Universal Robots PolyScope program: sand1.urp

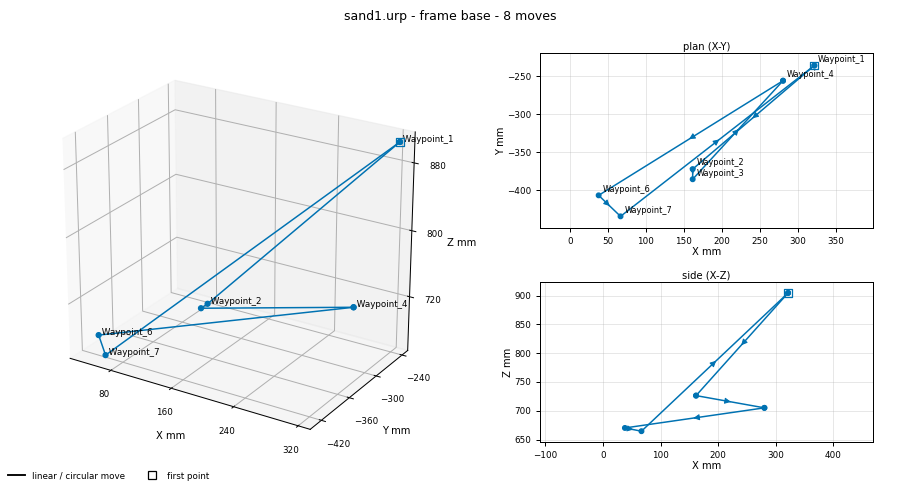
[picture p0: tool path of sand1.urp in frame base, 8 of 8 moves have a stored position in this frame; points joined in program order, loops and branches not executed]
Program sand1 (installation=default directory=/programs/archive createdIn=5.11.5.1010327 lastSavedIn=5.11.5.1010327 robotSerialNumber=20215500677)
Calibrated DH parameters: a=[0.000204, -0.239222, -0.391845, -0.000001, 0.000022, 0]; d=[0.162722, -355.808559, 353.37206, 2.570385, 0.099741, 0.099629]; alpha=[1.571124, 0.000988, 0.008295, 1.568963, -1.570303, 0]; deltaTheta=[0, -0.973091, 7.204745, 0.05153, 0, 0]
Robot Program (runOnlyOnce=true)
  MoveL speed 250 mm/s, acceleration 1200 mm/s^2 (useActiveTCP=true) feature=Base
    Waypoint Waypoint_1: TCP in base x=321.303 y=-235.884 z=904.602 mm, rx=1.6587 ry=-0.1473 rz=0.1861 rad; joints [-0.443, -84.298, -49.771, -109.018, 6.234, 255.071] deg
    Waypoint Waypoint_2: TCP in base x=161.455 y=-371.962 z=726.332 mm, rx=1.5708 ry=0 rz=0 rad; joints [-34.424, -75.969, -96.664, -7.98, 34.505, 180.726] deg
    Waypoint Waypoint_3: TCP in base x=161.455 y=-385.282 z=726.331 mm, rx=1.5708 ry=0 rz=0 rad; joints [-36.543, -77.681, -95.379, -7.51, 36.62, 180.691] deg
    SuppressedNode
      URCap Find Surface (Robotiq_Copilot, Robotiq Inc.) dataModel(NodeInitializedKey=true, WaitForSteadyWrenchOptionKey=false, ls_force=10.0, ls_distance=100.0, ls_speed=5.0, ls_if_distance=false, ls_if_force=false, ZeroSensorBeforeKey=true); state(isChildrenLocked=true)
        'Add Stop conditions from the Find Surface node'
    SuppressedNode
      Point_2 := Joint_6_nameget_actual_tcp_pose()
    URCap Finishing Tool Control (Robotiq_Copilot, Robotiq Inc.) dataModel(ToolOutputNameKey=digital_out[0], HackTriggeringContributionIsDefinedMethodKey=true)
    URCap Force Control (Robotiq_Copilot, Robotiq Inc.) dataModel(NodeInitializedKey=true, force_x=0, force_y=0, force_mx=0, force_my=0, force_mz=0, limit_x_neg=-100, limit_y_neg=-100, limit_z_neg=-100, limit_x_pos=100, limit_y_pos=100, limit_z_pos=100, limit_mx_neg=-20, limit_my_neg=-20, limit_mz_neg=-20, limit_mx_pos=20, limit_my_pos=20, limit_mz_pos=20, ft_control_x=false, ft_control_y=false, ft_control_mx=false, ft_control_my=false, ft_control_mz=false, stiffness_x=100, stiffness_y=100, stiffness_z_position=100, stiffness_mx=100, stiffness_my=100, stiffness_mz=100, adaptive_stiffness=true, ft_control_z=true, is_force_control_about_actual_position=true, force_z=2, HackTriggeringContributionIsDefinedMethodKey=true, TranslatableFeatureKey=1)
      URCap Force Event (Robotiq_Copilot, Robotiq Inc.) dataModel(NodeInitializedKey=true, NodeTitleKey=Force Event, InteractIfTimeoutOptionKey=false, InteractIfTimeoutNodeInsertedKey=false, InteractTimeoutKey=30, ForceReachedIfTimeoutOptionKey=false, ForceReachedIfTimeoutNodeInsertedKey=false, ForceReachedTimeoutKey=30, IfNotClickedOptionKey=false, IfNotClickedNodeInsertedKey=false, ForceDropRadioButtonKey=true, TorqueDropRadioButtonKey=false, ForceDropKey=10.0, TorqueDropKey=1.0, IsAddSingleTapButtonEnabledKey=true, IsAddDoubleTapButtonEnabledKey=true, AreDuplicatedTapNodesInTreeKey=false, SelectedForceEventKey=2, HackTriggeringContributionIsDefinedMethodKey=true); state(isChildrenLocked=true)
        'Wait until force and torque are reached.'
      URCap Multipoint Path (Robotiq_Copilot, Robotiq Inc.) dataModel(NodeInitializedKey=true, pathOptionsTypeKey=TOOL_ON_ROBOT, SPEED_VALUE=60, waypointIndexKey=6, OriginalFeatureAsArrayKey=[0.0, 0.0, 0.0, 0.0, 0.0, 0.0], offsetTypeKey=None, relativePathKey=false, HackTriggeringContributionIsDefinedMethodKey=true, urcapVersion=1.22.1)
        URCap Waypoint (Robotiq_Copilot, Robotiq Inc.) dataModel(NodeIndexKey=2, RenamedTitleKey=UnrenamedTitle, jointPositions=[-0.6336963823101671, -1.3523542565252598, -1.6673096435514436, -0.13197311436905323, 0.6350600830821999, 3.1537246700046184], waypointType=CURVE, waypointIndex=0, initialized=true, pose=[0.16146, -0.383763, 0.726308, 1.57082, -6.19253E-6, -1.9779E-5], urcapVersion=1.22.1)
        URCap Waypoint (Robotiq_Copilot, Robotiq Inc.) dataModel(NodeIndexKey=3, RenamedTitleKey=UnrenamedTitle, jointPositions=[-1.6957098491753975, -1.3658863619883306, -1.656896707797701, -0.11844284809070071, 1.6969853982500778, 3.1484054007216833], waypointType=LINE, waypointIndex=0, initialized=true, pose=[-0.170076, -0.383765, 0.726322, 1.5708, 9.0676E-6, 4.00998E-5], urcapVersion=1.22.1)
        URCap Waypoint (Robotiq_Copilot, Robotiq Inc.) dataModel(NodeIndexKey=4, RenamedTitleKey=UnrenamedTitle, jointPositions=[-1.694426789004269, -1.7628074068357105, -2.3522150592924156, 0.9733146680805841, 1.6877374087278332, 3.1446274473161964], waypointType=LINE, waypointIndex=0, initialized=true, pose=[-0.170098, -0.383754, 0.356007, 1.57074, -6.84536E-5, 2.60248E-5], urcapVersion=1.22.1)
        URCap Waypoint (Robotiq_Copilot, Robotiq Inc.) dataModel(NodeIndexKey=5, RenamedTitleKey=UnrenamedTitle, jointPositions=[-0.5963541519325757, -1.7728507109695997, -2.3383239441086037, 0.964207088945324, 0.5896524689063494, 3.1478558007161372], waypointType=LINE, waypointIndex=0, initialized=true, pose=[0.180447, -0.383757, 0.356019, 1.57073, -8.44249E-5, 5.93637E-5], urcapVersion=1.22.1)
        URCap Waypoint (Robotiq_Copilot, Robotiq Inc.) dataModel(jointPositions=[-0.5975693667723085, -1.3727915209140384, -1.7023849442810661, -0.07720128869267384, 0.5984260351890974, 3.154412409499461], waypointType=LINE, waypointIndex=0, initialized=true, NodeIndexKey=6, RenamedTitleKey=UnrenamedTitle, pose=[0.180407, -0.383745, 0.70645, 1.57073, -1.22865E-4, -1.7564E-5], urcapVersion=1.22.1)
        URCap Waypoint (Robotiq_Copilot, Robotiq Inc.) dataModel(NodeIndexKey=1, RenamedTitleKey=UnrenamedTitle, jointPositions=[-0.5171322037902302, -1.3116268501535489, -1.748472658069531, -0.09426390662152606, 0.518164482682443, 3.156107555249607], waypointType=LINE, waypointIndex=0, initialized=true, pose=[0.180457, -0.35571, 0.706455, 1.57075, -8.41481E-5, 1.43966E-5], urcapVersion=1.22.1)
    MoveL speed 250 mm/s, acceleration 1200 mm/s^2 (useActiveTCP=true) feature=Base
      Waypoint Waypoint_4: TCP in base x=280.164 y=-255.822 z=705.077 mm, rx=0 ry=0 rz=1.5708 rad; joints [-21.705, -98.483, -78.443, -273.101, 89.495, 201.626] deg; TCP offset x=0 y=0 z=0 mm, rx=0 ry=0 rz=0 rad
      Waypoint Waypoint_5: TCP in base x=280.159 y=-255.822 z=705.072 mm, rx=-2.1701 ry=0.1361 rz=-2.1395 rad; joints [-29.615, -75.15, -100.176, -5.412, 119.806, 277.278] deg
      Waypoint Waypoint_6: TCP in base x=37.925 y=-406.425 z=670.18 mm, rx=-2.1701 ry=0.1361 rz=-2.1395 rad; joints [-79.715, -88.983, -93.497, -0.043, 169.831, 274.895] deg
      Waypoint Waypoint_7: TCP in base x=66.67 y=-434.023 z=664.523 mm, rx=-2.1701 ry=0.1361 rz=-2.1395 rad; joints [-76.517, -92.59, -90.67, 1.319, 166.624, 275.512] deg
    URCap Force Control (Robotiq_Copilot, Robotiq Inc.) dataModel(NodeInitializedKey=true, force_x=0, force_y=0, force_mx=0, force_my=0, force_mz=0, limit_x_neg=-100, limit_y_neg=-100, limit_z_neg=-100, limit_x_pos=100, limit_y_pos=100, limit_z_pos=100, limit_mx_neg=-20, limit_my_neg=-20, limit_mz_neg=-20, limit_mx_pos=20, limit_my_pos=20, limit_mz_pos=20, ft_control_x=false, ft_control_y=false, ft_control_mx=false, ft_control_my=false, ft_control_mz=false, stiffness_x=100, stiffness_y=100, stiffness_z_position=100, stiffness_mx=100, stiffness_my=100, stiffness_mz=100, adaptive_stiffness=true, ft_control_z=true, is_force_control_about_actual_position=true, force_z=2, TranslatableFeatureKey=1, HackTriggeringContributionIsDefinedMethodKey=true)
      URCap Force Event (Robotiq_Copilot, Robotiq Inc.) dataModel(NodeInitializedKey=true, NodeTitleKey=Force Event, InteractIfTimeoutOptionKey=false, InteractIfTimeoutNodeInsertedKey=false, InteractTimeoutKey=30, ForceReachedIfTimeoutOptionKey=false, ForceReachedIfTimeoutNodeInsertedKey=false, ForceReachedTimeoutKey=30, IfNotClickedOptionKey=false, IfNotClickedNodeInsertedKey=false, ForceDropRadioButtonKey=true, TorqueDropRadioButtonKey=false, ForceDropKey=10.0, TorqueDropKey=1.0, IsAddSingleTapButtonEnabledKey=true, IsAddDoubleTapButtonEnabledKey=true, AreDuplicatedTapNodesInTreeKey=false, SelectedForceEventKey=2, HackTriggeringContributionIsDefinedMethodKey=true); state(isChildrenLocked=true)
        'Wait until force and torque are reached.'
      URCap Multipoint Path (Robotiq_Copilot, Robotiq Inc.) dataModel(NodeInitializedKey=true, pathOptionsTypeKey=TOOL_ON_ROBOT, SPEED_VALUE=60, waypointIndexKey=6, OriginalFeatureAsArrayKey=[0.0, 0.0, 0.0, 0.0, 0.0, 0.0], offsetTypeKey=None, relativePathKey=false, HackTriggeringContributionIsDefinedMethodKey=true, urcapVersion=1.22.1)
        URCap Waypoint (Robotiq_Copilot, Robotiq Inc.) dataModel(NodeIndexKey=2, RenamedTitleKey=UnrenamedTitle, pose=[0.06664663029983449, -0.434001461633361, 0.664540399037402, -2.1701126715242314, 0.136138147296733, -2.1394877884243306], jointPositions=[-1.335463359051822, -1.6159950132378471, -1.5825114514402818, 0.02305419155120525, 2.9081386184038664, 4.8086283127833], waypointType=CURVE, waypointIndex=0, initialized=true, urcapVersion=1.22.1)
        URCap Waypoint (Robotiq_Copilot, Robotiq Inc.) dataModel(NodeIndexKey=3, RenamedTitleKey=UnrenamedTitle, jointPositions=[-1.6957098491753975, -1.3658863619883306, -1.656896707797701, -0.11844284809070071, 1.6969853982500778, 3.1484054007216833], waypointType=LINE, waypointIndex=0, initialized=true, pose=[-0.170076, -0.383765, 0.726322, 1.5708, 9.0676E-6, 4.00998E-5], urcapVersion=1.22.1)
        URCap Waypoint (Robotiq_Copilot, Robotiq Inc.) dataModel(NodeIndexKey=4, RenamedTitleKey=UnrenamedTitle, jointPositions=[-1.694426789004269, -1.7628074068357105, -2.3522150592924156, 0.9733146680805841, 1.6877374087278332, 3.1446274473161964], waypointType=LINE, waypointIndex=0, initialized=true, pose=[-0.170098, -0.383754, 0.356007, 1.57074, -6.84536E-5, 2.60248E-5], urcapVersion=1.22.1)
        URCap Waypoint (Robotiq_Copilot, Robotiq Inc.) dataModel(NodeIndexKey=5, RenamedTitleKey=UnrenamedTitle, jointPositions=[-0.5963541519325757, -1.7728507109695997, -2.3383239441086037, 0.964207088945324, 0.5896524689063494, 3.1478558007161372], waypointType=LINE, waypointIndex=0, initialized=true, pose=[0.180447, -0.383757, 0.356019, 1.57073, -8.44249E-5, 5.93637E-5], urcapVersion=1.22.1)
        URCap Waypoint (Robotiq_Copilot, Robotiq Inc.) dataModel(jointPositions=[-0.5975693667723085, -1.3727915209140384, -1.7023849442810661, -0.07720128869267384, 0.5984260351890974, 3.154412409499461], waypointType=LINE, waypointIndex=0, initialized=true, NodeIndexKey=6, RenamedTitleKey=UnrenamedTitle, pose=[0.180407, -0.383745, 0.70645, 1.57073, -1.22865E-4, -1.7564E-5], urcapVersion=1.22.1)
        URCap Waypoint (Robotiq_Copilot, Robotiq Inc.) dataModel(NodeIndexKey=1, RenamedTitleKey=UnrenamedTitle, jointPositions=[-0.5171322037902302, -1.3116268501535489, -1.748472658069531, -0.09426390662152606, 0.518164482682443, 3.156107555249607], waypointType=LINE, waypointIndex=0, initialized=true, pose=[0.180457, -0.35571, 0.706455, 1.57075, -8.41481E-5, 1.43966E-5], urcapVersion=1.22.1)
    URCap Finishing Tool Control (Robotiq_Copilot, Robotiq Inc.) dataModel(FinishingToolStateKey=false, ToolOutputNameKey=digital_out[0], HackTriggeringContributionIsDefinedMethodKey=true)
    Waypoint Waypoint_1: TCP in base x=321.303 y=-235.884 z=904.602 mm, rx=1.6587 ry=-0.1473 rz=0.1861 rad; joints [-0.443, -84.298, -49.771, -109.018, 6.234, 255.071] deg
